FUNCTION_BLOCK FB_Raw_to_scaled
VAR_INPUT
	Value:REAL;
	Raw_min:REAL;
	Raw_max:REAL;
	Scaled_min:REAL;
	Scaled_max:REAL;
END_VAR
VAR_OUTPUT
	Scaled:REAL;
END_VAR
VAR
END_VAR

Raw_to_scaled();

METHOD Raw_to_scaled
VAR_INPUT
END_VAR
VAR_INST // added by the converter: edge detectors and wires of the graphical bodies
    _w1, _w3 : ANY;
    _w2 : REAL;
END_VAR
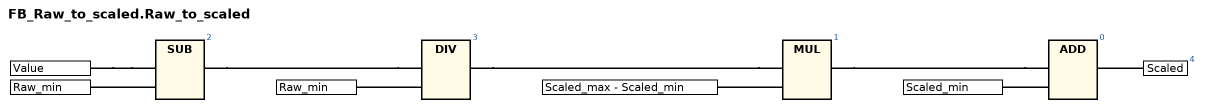
_w2 := _w1 + Scaled_min;
_w1 := _w3 * (Scaled_max - Scaled_min);
_w3 := (Value - Raw_min) / Raw_min;
Scaled := _w2;
END_METHOD

END_FUNCTION_BLOCK

(* stored: Version 1.1.0.1, ProductVersion 3.1.4024.0
   POU FB_Raw_to_scaled: Id {d214735a-a480-4ae2-bc21-7049593f3b3f}, SpecialFunc None
   Method Raw_to_scaled: Id {ab641ad7-b679-4a1a-8c6c-b4c8eb50fc66} *)
